# B&R Automation Studio project X20CP1382
Automation Studio 4.12.2.93; technology packages: mappView 5.16.1

## Configuration Config1

CPU X20CP1382, AutomationRuntime D4.83, Build 4.1.2, Safety 0.0, Vc V4.72.3

### Task classes (Cpu.sw)
```
Cyclic#4:
  Program1 <- Program1.prg
  Program <- Program.prg
  Zufall <- Zufall.prg
Binaries: FWRules, mvLoader, udbdef, TCData, iomap, sysconf, asfw, User, arconfig, ashwd, Role, ashwac
Libraries: standard, asieccon, astime, arssl, runtime, fileio
```

### Hardware
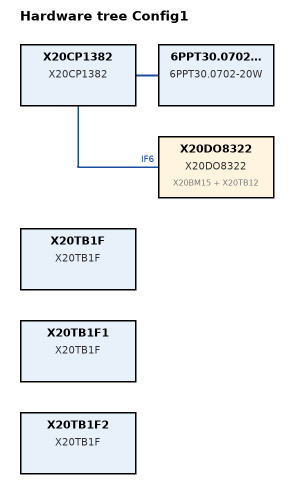
```
6PPT30.0702-20W : 6PPT30.0702-20W v1.3.5.0  [ETH1 -> X20CP1382.IF2 [Cable Type=PowerlinkCable, Length=10, Version=1.0.0.3]]
  Terminal = true
  Mode = Manual
  InternetAddress = 192.168.10.4
  Subnetmask = 255.255.255.0
  PasswordVNC = 
  PasswordCIFS = 
  PasswordService = 
  VncKeyMappingFile = VC\6PPT30.0702-20W.dis
X20BM15 : X20BM15 v1.1.0.0  [X2X1 -> X20CP1382.IF6 (NodeNumber=1)]
X20CP1382 : X20CP1382 v1.14.0.0  [X1 -> X1.SL; X2 -> X2.SL; X3 -> X3.SL]
  Module X1 (Type=X1, Virtual=true, Version=1.14.0.0)
    Connection (Connector=SS1, TargetModule=X20TB1F, TargetConnector=SS)
    Connection (Connector=SL, TargetModule=X20CP1382, TargetConnector=X1)
  Module X2 (Type=X2, Virtual=true, Version=1.14.0.0)
    Connection (Connector=SS1, TargetModule=X20TB1F1, TargetConnector=SS)
    Connection (Connector=SL, TargetModule=X20CP1382, TargetConnector=X2)
  Module X3 (Type=X3, Virtual=true, Version=1.14.0.0)
    Connection (Connector=SS1, TargetModule=X20TB1F2, TargetConnector=SS)
    Connection (Connector=SL, TargetModule=X20CP1382, TargetConnector=X3)
  Connector IF2:
    ActivateDevice = 1
    Mode = Manual
    InternetAddress = 192.168.10.5
    SubnetMask = 255.255.255.0
    ActivateSnmp = 2
  ConfigurationID = X20CP1382_Config1
  Simulation = 1
  ActivateOpcUa = 1
  OpcUaInformationModels_PV_Version = 1
X20DO8322 : X20DO8322 v1.5.0.0  [SS1 -> X20TB12a.SS; SL -> X20BM15.SL1]
X20TB12a : X20TB12 v1.0.0.0
X20TB1F : X20TB1F v1.0.0.0
X20TB1F1 : X20TB1F v1.0.0.0
X20TB1F2 : X20TB1F v1.0.0.0
```

### IoMap.iom - X20CP1382/IoMap.iom
```iecst
VAR_CONFIG
	::Program:directionThreadmillleft_DO AT %QX."X3".DigitalOutput12;
	::pumpeBig1_DO AT %QX."X3".DigitalOutput01;
	::pumpeBig2_DO AT %QX."X3".DigitalOutput02;
	::pumpeBig3_DO AT %QX."X3".DigitalOutput03;
	::pumpeBig4_DO AT %QX."X3".DigitalOutput04;
	::pumpeSmall1_DO AT %QX."X3".DigitalOutput05;
	::pumpeSmall2_DO AT %QX."X3".DigitalOutput06;
	::pumpeSmall3_DO AT %QX."X3".DigitalOutput07;
	::pumpeSmall4_DO AT %QX."X3".DigitalOutput08;
	::pumpeSmall5_DO AT %QX."X3".DigitalOutput09;
	::Program:directionTreadmillright_DO AT %QX."X3".DigitalOutput11;
	::pumpeSmall6_DO AT %QX."X3".DigitalOutput10;
	::Program:inductiveSensorBecherspender_DI AT %IX."X2".DigitalInput01;
	::Program:inductiveSensorEisstation_DI AT %IX."X2".DigitalInput02;
	::Program:inductiveSensorZitronenspende_DI AT %IX."X2".DigitalInput03;
	::Program:inductiveSensorCocktailmixer_DI AT %IX."X2".DigitalInput04;
	::Program:inductiveSensorBecherausgabe_DI AT %IX."X2".DigitalInput05;
	::Program:bechererkennungSpender_DI AT %IX."X2".DigitalInput06;
	::Program:bechererkennungAusgabe_DI AT %IX."X2".DigitalInput07;
	::Program:BecherspenderAktivieren_DO AT %QX."X20DO8322".DigitalOutput01;
	::Program:eisspenderAktivieren_DO AT %QX."X20DO8322".DigitalOutput02;
	::ERROR_DI AT %IX."X2".DigitalInput08 INVERSE;
	::Program:zitronenspenderAktivieren_DO AT %QX."X20DO8322".DigitalOutput03;
	::Program:lichtschrankeEismaschine_DI AT %IX."X2".DigitalInput10;
	::Program:endlagenschArmCocktailStation_DI AT %IX."X2".DigitalInput09;
	::Program:armCocktailstation_DO AT %QX."X20DO8322".DigitalOutput04;
END_VAR
```

## Logical view

### Global.var - Globale Variablen
```iecst
VAR
	pumpeBig1_DO : BOOL;
	pumpeBig2_DO : BOOL;
	pumpeBig3_DO : BOOL;
	pumpeBig4_DO : BOOL;
	pumpeSmall1_DO : BOOL;
	pumpeSmall2_DO : BOOL;
	pumpeSmall3_DO : BOOL;
	pumpeSmall4_DO : BOOL;
	pumpeSmall5_DO : BOOL;
	pumpeSmall6_DO : BOOL;
	cocktailFinished_var : BOOL;
	cocktailChosen_var : BOOL := FALSE; (*Gibt an, ob ein Cocktail gewählt wurde*)
	counterCocktailmixer_var : UDINT := 0; (*Wenn Station erstes mal angefahren wird Cocktail ausgegeben*)
	reingigunsmodus_var : BOOL := FALSE; (*Gibt an, ob die Reinigung aktiviert wurde*)
	cocktail_started : BOOL; (*Triggert die Pumpen für den aktuellen Cocktail*)
	ERROR_DI : BOOL := FALSE; (*STOPPT SPS KOMPLETT*)
	zufallscocktailAktivieren : BOOL;
	zutat_JaNein_ok : ARRAY[1..10] OF BOOL; (*Array mit Info, ob Zutat verwendet wird oder nicht*)
	zutat_Menge_ok : ARRAY[1..10] OF UINT; (*Array mit Info, wie viele ml der Zutat rein sollen*)
	zufallscocktail_var : BOOL := FALSE;
END_VAR
```

### Program Logical/Program (IEC)

#### Variables.var
```iecst
VAR
	armCocktailstation_DO : BOOL := FALSE; (*Gibt Signal für Arm nach oben und unten*)
	stationPercentage_var : USINT := 0; (*gibt in der Visualisierung den aktuellen Progress in % aus*)
	resetToStart_var : BOOL := TRUE; (*Fährt wieder an den Start*)
	passwordVisu_st : WSTRING[40] := "student"; (*Passwort 'student42'*)
	passwordVisuCorrect_var : BOOL := FALSE; (*gibt 1 aus wenn passwort stimmt*)
	lichtschrankeEismaschine_DI : BOOL := FALSE; (*Reagiert auf den Arduino mit der Lichtschranke*)
	inductiveSensorZitronenspende_DI : BOOL := FALSE; (*Station Zitronenspender Sensorerkennung*)
	inductiveSensorEisstation_DI : BOOL := FALSE; (*Station Eisstation Sensorerkennung*)
	inductiveSensorCocktailmixer_DI : BOOL := FALSE; (*Station Cocktailmixer Sensorenerkennung*)
	inductiveSensorBecherspender_DI : BOOL := FALSE; (*Station Becherspender Sensorerkennung*)
	inductiveSensorBecherausgabe_DI : BOOL := FALSE; (*Station Becherausgabe Sensorenerkennung*)
	hilfsDelayArmCocktailStation_var : UDINT := 0; (*hilft mit dem Timing für den Arm, damit die Pumpen sicher abgeschalten haben für bewegung*)
	resetCounter_var : USINT := 0; (*lässt wagen erstmal nach rechts und danach nach links fahren*)
	endlagenschArmCocktailStation_DI : BOOL := FALSE; (*Zeigt an, ob becher unter dem Endlagenschalter ist*)
	eisspenderAktivieren_DO : BOOL := FALSE; (*Aktiviert den Eisspender --> Arduino*)
	goToMainpage_var : BOOL := FALSE; (*Geht wieder zurück auf die Hauptseite*)
	directionThreadmill_right_var : BOOL := FALSE; (*Kann nur im Reinigunsprogramm gesetzt werden*)
	bechererkennungAusgabe_DI : BOOL := TRUE; (*Wenn endlageschalter nicht gedrückt ist, Becher entnommen*)
	bechererkennungSpender_DI : BOOL := FALSE; (*Wenn endlageschalter gedrückt, Becher in Halterung*)
	BecherspenderAktivieren_DO : BOOL := FALSE; (*Aktiviert Becherspender --> Arduino *)
	directionTreadmillright_DO : BOOL := FALSE; (*Steuert das Laufband nach rechts*)
	counterBecherspender_var : USINT := 0; (*Setzt die Zeit für die Sation Becherspender*)
	counterEisstation_var : UINT := 0; (*Setzt die Zeit für die Sation Eisstation*)
	counterBecherentnahme_var : USINT := 0; (*Setzt die Zeit für die Station Becherentnahme*)
	currentBecherausgabeState_var : USINT := 0; (*Switch Case Becherausgabe*)
	currentCocktialState_var : USINT := 0; (*Läuft die einzelnen unterstationen im Cocktailmixer ab*)
	currentStation_var : USINT := 0; (*Läuft die einzelnen Sationen ab*)
	delayCocktailStation_var : USINT := 0; (*Ein Delay nach dem Cocktaileinfüllen*)
	directionThreadmillleft_DO : BOOL := FALSE; (*Steuert das Laufband nach links*)
	directionThreadmill_left_var : BOOL := FALSE; (*Kann nur im Reinigunsprogramm gesetzt werden*)
	counterZitronenspender_var : USINT := 0; (*Setzt die Zeit für die Sation Zitronenspender*)
	zitronenspenderAktivieren_DO : BOOL := FALSE; (*Aktiviert Zitronenspender --> Arduino *)
END_VAR
VAR CONSTANT
	stationBecherentnahme_var : USINT := 4; (*Station Becherentnahme als Festwerte*)
	stationBecherspender_var : USINT := 0; (*Station Becherspender als Festwerte*)
	stationCocktailmixer_var : USINT := 3; (*Station Cocktailmixer als Festwerte*)
	stationEismaschine_var : USINT := 1; (*Station Eismaschine als Festwerte*)
END_VAR
VAR
	hilfsCounterEismaschine_var : UDINT := 0; (*Zählt einen Delay ein, damit der Wagen nicht direkt weiterfährt, wenn die Eiswürfel kommen*)
	deactivatesAllPumps_var : BOOL := FALSE; (*Kann im Reinigunsprogramm aktiviert werden und schaltet alle Pumpen AUS*)
	activatesAllPumps_var : BOOL := FALSE; (*Kann im Reinigungsprogramm aktiviert werden und schaltet alle Pumpen AN*)
END_VAR
VAR CONSTANT
	stationZitronenspender_var : USINT := 2; (*Station Zitronenspender als Festwert*)
END_VAR
```

#### Cyclic.st
```iecst
PROGRAM _CYCLIC
	// Visualisierungs Passworteingabe
	IF passwordVisu_st = "student42" THEN
		passwordVisuCorrect_var := TRUE;
	ELSE
		passwordVisuCorrect_var := FALSE;
	END_IF

	IF ERROR_DI = TRUE THEN
		// ON ERROR STOPPT ALLE PUMPEN DIREKT
		pumpeBig1_DO := FALSE;
		pumpeBig2_DO := FALSE;
		pumpeBig3_DO := FALSE;
		pumpeBig4_DO := FALSE;
		pumpeSmall1_DO := FALSE;
		pumpeSmall2_DO := FALSE;
		pumpeSmall3_DO := FALSE;
		pumpeSmall4_DO := FALSE;
		pumpeSmall5_DO := FALSE;
		pumpeSmall6_DO := FALSE;

		directionTreadmillright_DO := FALSE;
		directionThreadmillleft_DO := FALSE;
	ELSE
		// Reinigungsprogramm
		IF reingigunsmodus_var = TRUE THEN
			IF directionThreadmill_left_var = TRUE THEN
				directionThreadmillleft_DO := 0;
				directionTreadmillright_DO := 1;
			END_IF
			IF directionThreadmill_right_var = TRUE THEN
				directionThreadmillleft_DO := 1;
				directionTreadmillright_DO := 0;
			END_IF
			IF directionThreadmill_right_var = FALSE AND directionThreadmill_left_var = FALSE THEN
				directionThreadmillleft_DO := 0;
				directionTreadmillright_DO := 0;
			END_IF

			IF activatesAllPumps_var = TRUE THEN
				activatesAllPumps_var := FALSE;
				pumpeBig1_DO := TRUE;
				pumpeBig2_DO := TRUE;
				pumpeBig3_DO := TRUE;
				pumpeBig4_DO := TRUE;
				pumpeSmall1_DO := TRUE;
				pumpeSmall2_DO := TRUE;
				pumpeSmall3_DO := TRUE;
				pumpeSmall4_DO := TRUE;
				pumpeSmall5_DO := TRUE;
				pumpeSmall6_DO := TRUE;
			END_IF

			IF deactivatesAllPumps_var = TRUE THEN
				deactivatesAllPumps_var := FALSE;
				pumpeBig1_DO := FALSE;
				pumpeBig2_DO := FALSE;
				pumpeBig3_DO := FALSE;
				pumpeBig4_DO := FALSE;
				pumpeSmall1_DO := FALSE;
				pumpeSmall2_DO := FALSE;
				pumpeSmall3_DO := FALSE;
				pumpeSmall4_DO := FALSE;
				pumpeSmall5_DO := FALSE;
				pumpeSmall6_DO := FALSE;
			END_IF

		ELSE
			CASE currentStation_var OF
				stationBecherspender_var:
					// Setzt Website wieder auf Hauptseite nach erfolgten Durchlauf
					IF inductiveSensorBecherspender_DI = FALSE OR counterBecherspender_var > 0 THEN
						IF currentBecherausgabeState_var = 3 THEN
							goToMainpage_var := TRUE;
							resetCounter_var := 0;
							currentBecherausgabeState_var := 0;
						END_IF

						directionThreadmillleft_DO := 0;
						counterBecherentnahme_var := 0;
						IF cocktailChosen_var = TRUE THEN
							goToMainpage_var := FALSE;
							currentBecherausgabeState_var := 0;
							counterBecherspender_var := counterBecherspender_var + 1;

							stationPercentage_var := 10;

							IF counterBecherspender_var = 1 THEN
								BecherspenderAktivieren_DO := TRUE;
							ELSE
								BecherspenderAktivieren_DO := FALSE;
							END_IF

							IF bechererkennungSpender_DI = TRUE THEN
								directionTreadmillright_DO := 1;
								currentStation_var := currentStation_var + 1;
								BecherspenderAktivieren_DO := FALSE;
								stationPercentage_var := 20;
							END_IF
						END_IF
					END_IF

				stationEismaschine_var:
					IF inductiveSensorEisstation_DI = FALSE OR counterEisstation_var > 0 THEN
						directionTreadmillright_DO := 0;
						counterBecherspender_var := 0;
						counterEisstation_var := counterEisstation_var + 1;
						stationPercentage_var := 30;

						// 300 ms impuls for Arduino bei Anfahren der Station
						IF counterEisstation_var < 4 THEN
							eisspenderAktivieren_DO := TRUE;
						ELSE
							eisspenderAktivieren_DO := FALSE;
						END_IF

						// Wenn die Lichtschrankenrückmeldung kommt
						IF lichtschrankeEismaschine_DI = TRUE AND hilfsCounterEismaschine_var = 0 AND counterEisstation_var > 5 THEN
							hilfsCounterEismaschine_var := counterEisstation_var + 30;
						END_IF

						// Wenn der Wagen an der Station für 15 Sekunden steht oder das Signal vom Arduino kommt, das Lichtschranke ausgelöst wurde
						IF counterEisstation_var > 3000 OR hilfsCounterEismaschine_var <= counterEisstation_var AND hilfsCounterEismaschine_var <> 0 THEN
							directionTreadmillright_DO := 1;
							currentStation_var := currentStation_var + 1;
							stationPercentage_var := 40;
						END_IF
					END_IF

				stationZitronenspender_var:
					IF inductiveSensorZitronenspende_DI = FALSE OR counterZitronenspender_var > 0 THEN
						hilfsCounterEismaschine_var := 0;
						directionTreadmillright_DO := 0;
						counterEisstation_var := 0;
						counterZitronenspender_var := counterZitronenspender_var + 1;
						stationPercentage_var := 50;

						// 400 ms impuls for arduino
						IF counterZitronenspender_var < 4 THEN
							zitronenspenderAktivieren_DO := TRUE;
						ELSE
							zitronenspenderAktivieren_DO := FALSE;
						END_IF

						IF counterZitronenspender_var > 50 THEN
							directionTreadmillright_DO := 1;
							currentStation_var := currentStation_var + 1;
							stationPercentage_var := 60;
						END_IF
					END_IF

				stationCocktailmixer_var:
					IF inductiveSensorCocktailmixer_DI = FALSE OR counterCocktailmixer_var > 0 THEN
						directionTreadmillright_DO := 0;
						counterZitronenspender_var := 0;
						counterCocktailmixer_var := counterCocktailmixer_var + 1;

						CASE currentCocktialState_var OF
							0:
								// Arm fährt runter --> Signal Arduino
								IF counterCocktailmixer_var > 3 THEN
									armCocktailstation_DO := TRUE;
									currentCocktialState_var := currentCocktialState_var + 1;
									stationPercentage_var := 70;
								END_IF
							1:
								// Setzt Arduino Signal wieder auf 0
								IF counterCocktailmixer_var > 7 THEN;
									armCocktailstation_DO := FALSE;
									currentCocktialState_var := currentCocktialState_var + 1;
								END_IF

							2:
								// Startet Cocktail, wenn Endlagenschalter Anschlägt
								IF counterCocktailmixer_var >= 30 AND endlagenschArmCocktailStation_DI = TRUE THEN
									cocktail_started := FALSE;
									currentCocktialState_var := currentCocktialState_var + 1;
								END_IF
							3:
								//	IF cocktailFinished_var = TRUE THEN
								IF counterCocktailmixer_var >= 50 AND pumpeBig1_DO = 0 AND pumpeBig2_DO = 0 AND pumpeBig3_DO = 0 AND pumpeBig4_DO = 0 AND pumpeSmall1_DO = 0 AND pumpeSmall2_DO = 0 AND pumpeSmall3_DO = 0 AND pumpeSmall4_DO = 0 AND  pumpeSmall5_DO = 0 AND  pumpeSmall6_DO = 0 THEN
									stationPercentage_var := 80;
									cocktailFinished_var := TRUE;

									hilfsDelayArmCocktailStation_var := counterCocktailmixer_var + 5;
									currentCocktialState_var := currentCocktialState_var + 1;
								END_IF
							4:
								// Delay nach dem die Pumpen abgeschalten haben 500ms
								IF counterCocktailmixer_var >= hilfsDelayArmCocktailStation_var AND armCocktailstation_DO = FALSE THEN
									armCocktailstation_DO := TRUE;
									hilfsDelayArmCocktailStation_var :=  counterCocktailmixer_var + 4;
									currentCocktialState_var := currentCocktialState_var + 1;
								END_IF
							5:
								// 400 ms Signal auf den Ausgang beenden
								IF counterCocktailmixer_var >= hilfsDelayArmCocktailStation_var AND armCocktailstation_DO = TRUE THEN
									stationPercentage_var := 90;
									armCocktailstation_DO := FALSE;
									hilfsDelayArmCocktailStation_var := counterCocktailmixer_var + 16;
									currentCocktialState_var := currentCocktialState_var + 1;
								END_IF
							6:
								// geht zur nächsten Station nachdem der arm 1.6 Sekunden Zeit hatte hochzufahren
								IF 	counterCocktailmixer_var >= hilfsDelayArmCocktailStation_var AND stationPercentage_var = 90 THEN
									directionTreadmillright_DO := TRUE;
									currentStation_var := currentStation_var + 1;
									currentCocktialState_var := 0;
								END_IF
						END_CASE
					END_IF

				stationBecherentnahme_var:
					CASE currentBecherausgabeState_var OF
						0: // Stoppt an Station
							IF inductiveSensorBecherausgabe_DI = FALSE OR bechererkennungAusgabe_DI = TRUE THEN
								counterCocktailmixer_var := 0;
								currentBecherausgabeState_var := 1;
								cocktailFinished_var := 0;
								stationPercentage_var := 100;
								directionTreadmillright_DO := 0;
								delayCocktailStation_var := 0;
							END_IF

						1:// Wenn Becher steht
							// drei Sekunden verzögerung zum verlässlichen erkennen des Endlagenschalters
							IF counterBecherentnahme_var >= 30 THEN
								// Erkennt wenn Becher Ausgegeben wurde --> Wird als zweites ausgeführt
								IF bechererkennungAusgabe_DI = FALSE THEN
									currentBecherausgabeState_var := 2;
								END_IF
							ELSE
								counterBecherentnahme_var := counterBecherentnahme_var + 1;
							END_IF

						2:
							// Zählt Für Verzögerung beim herausnehmen
							IF counterBecherentnahme_var > 0 THEN
								counterBecherentnahme_var := counterBecherentnahme_var + 1;
							END_IF

							// Fährt mit verzögerung wieder zum Start
							IF counterBecherentnahme_var >= 60 THEN
								directionTreadmillright_DO := 0;
								directionThreadmillleft_DO := 1;
								currentStation_var := 0;
								cocktailChosen_var := FALSE;
								currentBecherausgabeState_var := 3;
							END_IF
					END_CASE
			END_CASE
		END_IF

		// Zurücksetzen auf Start
		IF resetToStart_var = TRUE THEN
			IF resetCounter_var < 10 THEN
				resetCounter_var := resetCounter_var + 1;
				pumpeBig1_DO := FALSE;
				pumpeBig2_DO := FALSE;
				pumpeBig3_DO := FALSE;
				pumpeBig4_DO := FALSE;
				pumpeSmall1_DO := FALSE;
				pumpeSmall2_DO := FALSE;
				pumpeSmall3_DO := FALSE;
				pumpeSmall4_DO := FALSE;
				pumpeSmall5_DO := FALSE;
				pumpeSmall6_DO := FALSE;

				counterBecherspender_var := 0;
				counterEisstation_var := 0;
				counterZitronenspender_var := 0;
				counterCocktailmixer_var := 0;

				directionThreadmillleft_DO := 0;

				// Fährt nich weiter, wenn hinten der Taster gedrückt wird
				IF bechererkennungAusgabe_DI = FALSE THEN
					directionTreadmillright_DO := 1;
				ELSE
					directionTreadmillright_DO := 0;
				END_IF
			ELSE
				directionTreadmillright_DO := 0;
				currentStation_var := 4;
				currentBecherausgabeState_var := 2;
				counterBecherentnahme_var := 100;

				resetToStart_var := FALSE;
			END_IF
		END_IF
	END_IF
END_PROGRAM
```

#### Init.st
```iecst
PROGRAM _INIT

END_PROGRAM
```

### Program Logical/Program1 (IEC)

#### Types.typ
```iecst
TYPE
	cocktail_name :
		(
		wodka_cola,
		kirschcola,
		testcocktail,
		wodka_osaft,
		gruenewiese,
		angelblue,
		brassmonkey,
		kiba,
		rumcola,
		gintonic,
		bluelagoon,
		cola,
		osaft,
		banane,
		tonic,
		sprite,
		zufallscocktail
		);
END_TYPE
```

#### Variables.var
```iecst
VAR
	cocktail_var : cocktail_name;
	cocktail_start : BOOL;
	TOF_01 : TOF;
	TOF_02 : TOF;
	TOF_03 : TOF;
	TOF_04 : TOF;
	TOF_05 : TOF;
	TOF_06 : TOF;
	TOF_07 : TOF;
	TOF_08 : TOF;
	TOF_09 : TOF;
	TOF_10 : TOF;
	pumptime_01 : TIME;
	pumptime_02 : TIME;
	pumptime_03 : TIME;
	pumptime_04 : TIME;
	pumptime_05 : TIME;
	pumptime_06 : TIME;
	pumptime_07 : TIME;
	pumptime_08 : TIME;
	pumptime_09 : TIME;
	pumptime_10 : TIME;
	ml_wodkacola_wodka : UINT := 50;
	ml_wodkacola_cola : UINT := 250;
	ml_wodkaosaft_osaft : UINT := 250;
	ml_wodkaosaft_wodka : UINT := 50;
	ml_rumcola_cola : UINT := 250;
	ml_rumcola_rum : UINT := 50;
	ml_kirschcola_cola : UINT := 210;
	ml_kirschcola_kirsch : UINT := 90;
	ml_gruenewiese_osaft : UINT := 220;
	ml_gruenewiese_bc : UINT := 80;
	ml_angelblue_sprite : UINT := 200;
	ml_angelblue_bc : UINT := 70;
	ml_angelblue_wodka : UINT := 30;
	ml_brassmonkey_osaft : UINT := 240;
	ml_brassmonkey_wodka : UINT := 30;
	ml_brassmonkey_rum : UINT := 30;
	ml_kiba_banane : UINT := 210;
	ml_kiba_kirsch : UINT := 90;
	ml_gintonic_tonic : UINT := 250;
	ml_gintonic_gin : UINT := 50;
	ml_osaft : UINT := 300;
	ml_cola : UINT := 300;
	ml_banane : UINT := 300;
	ml_tonic : UINT := 300;
	ml_sprite : UINT := 300;
	ml_bluelagoon_sprite : UINT := 220;
	ml_bluelagoon_bc : UINT := 80;
	wodka_cola_var : BOOL := FALSE;
	kirschcola_var : BOOL := FALSE;
	testcocktail_var : BOOL := FALSE;
	gruenewiese_var : BOOL := FALSE;
	brassmonkey_var : BOOL := FALSE;
	angelblue_var : BOOL := FALSE;
	kiba_var : BOOL := FALSE;
	rumcola_var : BOOL := FALSE;
	gintonic_var : BOOL := FALSE;
	wodka_osaft_var : BOOL := FALSE;
	osaft_var : BOOL := FALSE;
	cola_var : BOOL := FALSE;
	banane_var : BOOL := FALSE;
	tonic_var : BOOL := FALSE;
	sprite_var : BOOL := FALSE;
	bluelagoon_var : BOOL := FALSE;
END_VAR
VAR RETAIN
	Anzahl_Cocktails : ARRAY[0..19] OF INT := [20(0)];
END_VAR
```

#### Cyclic.st
```iecst
PROGRAM _CYCLIC

	IF (cocktail_start = FALSE AND cocktail_started = FALSE) THEN
		cocktail_start := TRUE;
	END_IF

	// Wenn Reinigungsprogramm aktiviert ist, soll kein Cocktail gemacht werden
	IF reingigunsmodus_var = FALSE AND ERROR_DI = FALSE THEN
		CASE cocktail_var OF
			wodka_cola:
				pumptime_01 :=	UINT_TO_TIME(ml_wodkacola_cola)*108;
				pumptime_02 :=	UINT_TO_TIME(ml_wodkacola_wodka)*330;

				TOF_01(IN:= cocktail_start , PT:= pumptime_01 );
				pumpeBig2_DO:=TOF_01.Q;

				TOF_02(IN:= cocktail_start , PT:= pumptime_02 );
				pumpeSmall3_DO:=TOF_02.Q;

			rumcola:
				pumptime_01 :=	UINT_TO_TIME(ml_rumcola_cola)*108;
				pumptime_02 :=	UINT_TO_TIME(ml_rumcola_rum)*420;

				TOF_01(IN:= cocktail_start , PT:= pumptime_01 );
				pumpeBig2_DO:=TOF_01.Q;

				TOF_02(IN:= cocktail_start , PT:= pumptime_02 );
				pumpeSmall2_DO:=TOF_02.Q;

			kirschcola:
				pumptime_01 :=	UINT_TO_TIME(ml_kirschcola_cola)*108;
				pumptime_02 :=	UINT_TO_TIME(ml_kirschcola_kirsch)*390;

				TOF_01(IN:= cocktail_start , PT:= pumptime_01 );
				pumpeBig2_DO:=TOF_01.Q;

				TOF_02(IN:= cocktail_start , PT:= pumptime_02 );
				pumpeSmall5_DO:=TOF_02.Q;

			gruenewiese:
				pumptime_01 :=	UINT_TO_TIME(ml_gruenewiese_osaft)*118;
				pumptime_02 :=	UINT_TO_TIME(ml_gruenewiese_bc)*350;

				TOF_01(IN:= cocktail_start , PT:= pumptime_01 );
				pumpeBig4_DO:=TOF_01.Q;

				TOF_02(IN:= cocktail_start , PT:= pumptime_02 );
				pumpeSmall6_DO:=TOF_02.Q;

			angelblue:
				pumptime_01 :=	UINT_TO_TIME(ml_angelblue_sprite)*111;
				pumptime_02 :=	UINT_TO_TIME(ml_angelblue_bc)*350;
				pumptime_03 := UINT_TO_TIME(ml_angelblue_wodka)*330;

				TOF_01(IN:= cocktail_start , PT:= pumptime_01 );
				pumpeBig1_DO:=TOF_01.Q;

				TOF_02(IN:= cocktail_start , PT:= pumptime_02 );
				pumpeSmall6_DO:=TOF_02.Q;

				TOF_03(IN:= cocktail_start , PT:= pumptime_03 );
				pumpeSmall3_DO:=TOF_03.Q;

			brassmonkey:
				pumptime_01 :=	UINT_TO_TIME(ml_brassmonkey_osaft)*118;
				pumptime_02 :=	UINT_TO_TIME(ml_brassmonkey_rum)*420;
				pumptime_03 := UINT_TO_TIME(ml_angelblue_wodka)*330;

				TOF_01(IN:= cocktail_start , PT:= pumptime_01 );
				pumpeBig4_DO:=TOF_01.Q;

				TOF_02(IN:= cocktail_start , PT:= pumptime_02 );
				pumpeSmall2_DO:=TOF_02.Q;

				TOF_03(IN:= cocktail_start , PT:= pumptime_03 );
				pumpeSmall3_DO:=TOF_03.Q;

			wodka_osaft:
				pumptime_01 :=	UINT_TO_TIME(ml_wodkaosaft_osaft)*118;
				pumptime_02 :=	UINT_TO_TIME(ml_wodkaosaft_wodka)*330;

				TOF_01(IN:= cocktail_start , PT:= pumptime_01 );
				pumpeBig4_DO:=TOF_01.Q;

				TOF_02(IN:= cocktail_start , PT:= pumptime_02 );
				pumpeSmall3_DO:=TOF_02.Q;

			testcocktail:
				pumptime_01 :=	T#2s;
				pumptime_02 :=	T#2s;

				TOF_01(IN:= cocktail_start , PT:= pumptime_01 );
				pumpeBig4_DO:=TOF_01.Q;

				TOF_02(IN:= cocktail_start , PT:= pumptime_02 );
				pumpeSmall3_DO:=TOF_02.Q;

			kiba:
				pumptime_01 :=	UINT_TO_TIME(ml_kiba_banane)*105;
				pumptime_02 :=	UINT_TO_TIME(ml_kiba_kirsch)*390;

				TOF_01(IN:= cocktail_start , PT:= pumptime_01 );
				pumpeBig3_DO:=TOF_01.Q;

				TOF_02(IN:= cocktail_start , PT:= pumptime_02 );
				pumpeSmall5_DO:=TOF_02.Q;

			gintonic:
				pumptime_01 :=	UINT_TO_TIME(ml_gintonic_tonic)*390;
				pumptime_02 :=	UINT_TO_TIME(ml_gintonic_gin)*300;

				TOF_01(IN:= cocktail_start , PT:= pumptime_01 );
				pumpeSmall1_DO:=TOF_01.Q;

				TOF_02(IN:= cocktail_start , PT:= pumptime_02 );
				pumpeSmall4_DO:=TOF_02.Q;

			bluelagoon:
				pumptime_01 :=	UINT_TO_TIME(ml_bluelagoon_sprite)*111;
				pumptime_02 :=	UINT_TO_TIME(ml_bluelagoon_bc)*350;

				TOF_01(IN:= cocktail_start , PT:= pumptime_01 );
				pumpeBig1_DO:=TOF_01.Q;

				TOF_02(IN:= cocktail_start , PT:= pumptime_02 );
				pumpeSmall6_DO:=TOF_02.Q;

			zufallscocktail:
				pumptime_01 :=	UINT_TO_TIME(zutat_Menge_ok[1])*111;
				pumptime_02 :=	UINT_TO_TIME(zutat_Menge_ok[2])*108;
				pumptime_03 :=	UINT_TO_TIME(zutat_Menge_ok[3])*105;
				pumptime_02 :=	UINT_TO_TIME(zutat_Menge_ok[4])*118;
				pumptime_05 :=	UINT_TO_TIME(zutat_Menge_ok[5])*390;
				pumptime_06 :=	UINT_TO_TIME(zutat_Menge_ok[6])*420;
				pumptime_07 :=	UINT_TO_TIME(zutat_Menge_ok[7])*330;
				pumptime_08 :=	UINT_TO_TIME(zutat_Menge_ok[8])*300;
				pumptime_09 :=	UINT_TO_TIME(zutat_Menge_ok[9])*390;
				pumptime_10 :=	UINT_TO_TIME(zutat_Menge_ok[10])*350;

				IF zutat_JaNein_ok[1] = TRUE THEN
					TOF_01(IN:= cocktail_start , PT:= pumptime_01 );
					pumpeBig1_DO:=TOF_01.Q;
				END_IF
				IF zutat_JaNein_ok[2] = TRUE THEN
					TOF_02(IN:= cocktail_start , PT:= pumptime_02 );
					pumpeBig2_DO:=TOF_02.Q;
				END_IF
				IF zutat_JaNein_ok[3] = TRUE THEN
					TOF_03(IN:= cocktail_start , PT:= pumptime_03 );
					pumpeBig3_DO:=TOF_03.Q;
				END_IF
				IF zutat_JaNein_ok[4] = TRUE THEN
					TOF_04(IN:= cocktail_start , PT:= pumptime_04 );
					pumpeBig4_DO:=TOF_04.Q;
				END_IF
				IF zutat_JaNein_ok[5] = TRUE THEN
					TOF_05(IN:= cocktail_start , PT:= pumptime_05 );
					pumpeSmall1_DO:=TOF_05.Q;
				END_IF
				IF zutat_JaNein_ok[6] = TRUE THEN
					TOF_06(IN:= cocktail_start , PT:= pumptime_06 );
					pumpeSmall2_DO:=TOF_06.Q;
				END_IF
				IF zutat_JaNein_ok[7] = TRUE THEN
					TOF_07(IN:= cocktail_start , PT:= pumptime_07 );
					pumpeSmall3_DO:=TOF_07.Q;
				END_IF
				IF zutat_JaNein_ok[8] = TRUE THEN
					TOF_08(IN:= cocktail_start , PT:= pumptime_08 );
					pumpeSmall4_DO:=TOF_08.Q;
				END_IF
				IF zutat_JaNein_ok[9] = TRUE THEN
					TOF_09(IN:= cocktail_start , PT:= pumptime_09 );
					pumpeSmall5_DO:=TOF_09.Q;
				END_IF
				IF zutat_JaNein_ok[10] = TRUE THEN
					TOF_10(IN:= cocktail_start , PT:= pumptime_10 );
					pumpeSmall6_DO:=TOF_10.Q;
				END_IF

			osaft:
				pumptime_01 :=	UINT_TO_TIME(ml_osaft)*118;

				TOF_01(IN:= cocktail_start , PT:= pumptime_01 );
				pumpeBig4_DO:=TOF_01.Q;
			cola:
				pumptime_01 :=	UINT_TO_TIME(ml_cola)*108;

				TOF_01(IN:= cocktail_start , PT:= pumptime_01 );
				pumpeBig2_DO:=TOF_01.Q;
			banane:
				pumptime_01 :=	UINT_TO_TIME(ml_banane)*105;

				TOF_01(IN:= cocktail_start , PT:= pumptime_01 );
				pumpeBig3_DO:=TOF_01.Q;
			tonic:
				pumptime_01 :=	UINT_TO_TIME(ml_tonic)*390;

				TOF_01(IN:= cocktail_start , PT:= pumptime_01 );
				pumpeSmall1_DO:=TOF_01.Q;
			sprite:
				pumptime_01 :=	UINT_TO_TIME(ml_sprite)*111;

				TOF_01(IN:= cocktail_start , PT:= pumptime_01 );
				pumpeBig1_DO:=TOF_01.Q;

		END_CASE
	END_IF
	// IF Cocktail was chosen in the visualisation --> Cocktailchosen == True
	IF wodka_cola_var = 1 OR kirschcola_var = 1 OR testcocktail_var = 1 OR wodka_osaft_var = 1 OR gruenewiese_var = 1 OR angelblue_var = 1 OR brassmonkey_var = 1 OR kiba_var = 1 OR rumcola_var = 1 OR gintonic_var = 1 OR bluelagoon_var = 1 OR osaft_var = 1 OR cola_var = 1 OR banane_var = 1 OR tonic_var = 1 OR sprite_var = 1 OR zufallscocktail_var = 1 THEN
		cocktailChosen_var := TRUE;
	END_IF

	IF (cocktail_start = TRUE AND cocktail_started = FALSE) THEN
		cocktail_start := FALSE;
		cocktail_started := TRUE;

		// Variable, dass Cocktail beendet wurde
		cocktailFinished_var := TRUE;
	END_IF

	// Setzt den Schalter zurück
	IF wodka_cola_var = TRUE THEN
		cocktail_var := wodka_cola;
		wodka_cola_var := FALSE;
		Anzahl_Cocktails [wodka_cola] := Anzahl_Cocktails [wodka_cola] + 1;
	END_IF
	IF kirschcola_var = TRUE THEN
		cocktail_var := kirschcola;
		kirschcola_var := FALSE;
		Anzahl_Cocktails [kirschcola] := Anzahl_Cocktails [kirschcola] + 1;
	END_IF
	IF testcocktail_var = TRUE THEN
		cocktail_var := testcocktail;
		testcocktail_var := FALSE;
		Anzahl_Cocktails [testcocktail] := Anzahl_Cocktails [testcocktail] + 1;
	END_IF
	IF wodka_osaft_var = TRUE THEN
		cocktail_var := wodka_osaft;
		wodka_osaft_var := FALSE;
		Anzahl_Cocktails [wodka_osaft] := Anzahl_Cocktails [wodka_osaft] + 1;
	END_IF
	IF gruenewiese_var = TRUE THEN
		cocktail_var := gruenewiese;
		gruenewiese_var := FALSE;
		Anzahl_Cocktails [gruenewiese] := Anzahl_Cocktails [gruenewiese] + 1;
	END_IF
	IF angelblue_var = TRUE THEN
		cocktail_var := angelblue;
		angelblue_var := FALSE;
		Anzahl_Cocktails [angelblue] := Anzahl_Cocktails [angelblue] + 1;
	END_IF
	IF brassmonkey_var = TRUE THEN
		cocktail_var := brassmonkey;
		brassmonkey_var := FALSE;
		Anzahl_Cocktails [brassmonkey] := Anzahl_Cocktails [brassmonkey] + 1;
	END_IF
	IF kiba_var = TRUE THEN
		cocktail_var := kiba;
		kiba_var := FALSE;
		Anzahl_Cocktails [kiba] := Anzahl_Cocktails [kiba] + 1;
	END_IF
	IF rumcola_var = TRUE THEN
		cocktail_var := rumcola;
		rumcola_var := FALSE;
		Anzahl_Cocktails [rumcola] := Anzahl_Cocktails [rumcola] + 1;
	END_IF
	IF gintonic_var = TRUE THEN
		cocktail_var := gintonic;
		gintonic_var := FALSE;
		Anzahl_Cocktails [gintonic] := Anzahl_Cocktails [gintonic] + 1;
	END_IF
	IF bluelagoon_var = TRUE THEN
		cocktail_var := bluelagoon;
		bluelagoon_var := FALSE;
		Anzahl_Cocktails [bluelagoon] := Anzahl_Cocktails [bluelagoon] + 1;
	END_IF
	IF osaft_var = TRUE THEN
		cocktail_var := osaft;
		osaft_var := FALSE;
		Anzahl_Cocktails [osaft] := Anzahl_Cocktails [osaft] + 1;
	END_IF
	IF cola_var = TRUE THEN
		cocktail_var := cola;
		cola_var := FALSE;
		Anzahl_Cocktails [cola] := Anzahl_Cocktails [cola] + 1;
	END_IF
	IF banane_var = TRUE THEN
		cocktail_var := banane;
		banane_var := FALSE;
		Anzahl_Cocktails [banane] := Anzahl_Cocktails [banane] + 1;
	END_IF
	IF tonic_var = TRUE THEN
		cocktail_var := tonic;
		tonic_var := FALSE;
		Anzahl_Cocktails [tonic] := Anzahl_Cocktails [tonic] + 1;
	END_IF
	IF sprite_var = TRUE THEN
		cocktail_var := sprite;
		sprite_var := FALSE;
		Anzahl_Cocktails [sprite] := Anzahl_Cocktails [sprite] + 1;
	END_IF
	IF zufallscocktail_var = TRUE THEN
		cocktail_var := zufallscocktail;
		zufallscocktail_var := FALSE;
		Anzahl_Cocktails [zufallscocktail] := Anzahl_Cocktails [zufallscocktail] + 1;
	END_IF
END_PROGRAM
```

#### Init.st
```iecst
PROGRAM _INIT
	cocktail_started := TRUE;

	cocktail_var := 0;
END_PROGRAM
```

- Visualisation Logical/mappView (not shown)

### Program Logical/Zufall (IEC)

#### Variables.var
```iecst
VAR
	Random_Number : ARRAY[1..20] OF USINT; (*Array der Zufallszahlen*)
	m : USINT; (*Hilfsvariable*)
	i : USINT; (*Hilfsvariable*)
	Number_Counter : ARRAY[1..10] OF USINT; (*Zählt, wie oft die Zutaten jeweils vertreten sind*)
	zutat_Menge : ARRAY[1..10] OF UINT;
	zutat_JaNein : ARRAY[1..10] OF BOOL;
	ml : USINT;
	cycle_counter : LREAL; (*Anzahl der durchlaufenen Zyklen zählen*)
	access_counter : USINT; (*Kontrollvariable für Tests, Zählt Anzahl Zugriffe auf Mengenarray bei Mengenbestimmung*)
	k : USINT; (*Hilfsvariable*)
	n : USINT; (*Hilfsvariable*)
	p : USINT; (*Hilfsvariable*)
	q : USINT; (*Hilfsvariable*)
	r : USINT; (*Hilfsvariable*)
	ml_ausgabe : UINT; (*Nur Informationsvariable, um zu testen, wieviele ml am ende tatsächlich rauskommen*)
	menge_alkohol : UINT; (*zum Filtern von Ausreißern*)
	menge_alkoholfrei : UINT; (*zum Filtern von Ausreißern*)
END_VAR
```

#### Cyclic.st
```iecst
PROGRAM _CYCLIC
	IF zufallscocktail_var = FALSE THEN
			//willkürliches Verrechnen zum Erstellen eines Zufalls
			Random_Number[01] := (Random_Number[01] + 73) * ((Random_Number[17] + 1) MOD 14);
			Random_Number[02] := (Random_Number[09] + 73) * ((Random_Number[12] + 1) MOD 16);
			Random_Number[03] := (Random_Number[13] + 73) * ((Random_Number[20] + 1) MOD 11);
			Random_Number[04] := (Random_Number[18] + 73) * ((Random_Number[09] + 1) MOD 17);
			Random_Number[05] := (Random_Number[08] + 73) * ((Random_Number[16] + 1) MOD 19);
			Random_Number[06] := (Random_Number[20] + 72) * ((Random_Number[09] + 1) MOD 13);
			Random_Number[07] := (Random_Number[07] + 73) * ((Random_Number[01] + 1) MOD 17);
			Random_Number[08] := (Random_Number[11] + 73) * ((Random_Number[18] + 1) MOD 18);
			Random_Number[09] := (Random_Number[19] + 73) * ((Random_Number[12] + 1) MOD 11);
			Random_Number[10] := (Random_Number[12] + 73) * ((Random_Number[07] + 1) MOD 16);
			Random_Number[11] := (Random_Number[04] + 73) * ((Random_Number[02] + 1) MOD 10);
			Random_Number[12] := (Random_Number[03] + 73) * ((Random_Number[10] + 1) MOD 19);
			Random_Number[13] := (Random_Number[16] + 73) * ((Random_Number[15] + 1) MOD 18);
			Random_Number[14] := (Random_Number[06] + 73) * ((Random_Number[14] + 1) MOD 17);
			Random_Number[15] := (Random_Number[15] + 73) * ((Random_Number[04] + 1) MOD 15);
			Random_Number[16] := (Random_Number[05] + 73) * ((Random_Number[05] + 1) MOD 10);
			Random_Number[17] := (Random_Number[10] + 73) * ((Random_Number[06] + 1) MOD 18);
			Random_Number[18] := (Random_Number[14] + 73) * ((Random_Number[03] + 1) MOD 14);
			Random_Number[19] := (Random_Number[17] + 73) * ((Random_Number[19] + 1) MOD 19);
			Random_Number[20] := (Random_Number[02] + 73) * ((Random_Number[11] + 1) MOD 16);
			// MOD2: Durchschnittlich 2,6 Zutaten pro Cocktail
			FOR i := 1 TO 4 DO		//Zutatjanein setzen für nicht-alkoholische, Zählen
				IF Random_Number[i] MOD 3 = 0 THEN	//durch MOD 2 häufiger als alkoholische
					zutat_JaNein[i] := TRUE;
					Number_Counter[i] := Number_Counter[i] + 1;
				ELSE
					zutat_JaNein[i] := FALSE;
				END_IF
			END_FOR;
			// MOD4: Durchschnittlich 2,6 Zutaten pro Cocktail
			FOR i := 5 TO 10 DO		//Zutatjanein setzen für alkoholische, Zählen
				IF Random_Number[i] MOD 7 = 0 THEN		//durch MOD 4 weniger häufig als nich-alkoholische
					zutat_JaNein[i] := TRUE;
					Number_Counter[i] := Number_Counter[i] + 1;
				ELSE
					zutat_JaNein[i] := FALSE;
				END_IF
			END_FOR;

			ml := 30;		//Menge zurücksetzen
			ml_ausgabe := 0; //Ausgabemenge zurücksetzen
			FOR i := 1 TO 10 DO		//Mengenarray zurücksetzen
				zutat_Menge[i] := 0;
			END_FOR;

			REPEAT 			//Festlegen der Getränkemengen, zweimal durchgehen
				//über Modulo Werte aufnehmen, Multiplizieren und in zutat_Menge Array schreiben
				IF n MOD 2 = 0 THEN		//es wird immer zwischen den einstelligen und zweistelligen Zufallszahlen gewechselt
					p := 10;
				ELSIF n MOD 3 = 0 THEN
					r := 87;		//alles mit r ist nur, um etwas mehr Zufall zu erzeugen
				ELSE
					p := 0;
					r := 0;
				END_IF
				//Mengen durch unterschiedliche Modulo unterschiedlich festlegen
				FOR i := 1 TO 4 DO
					IF zutat_JaNein[i] = TRUE THEN
						//	m := ml/2;		//m enthält Anteil, der noch aufgefüllt werden muss, hier kann durchschnittliche Menge angepasst werden
						k := (Random_Number[i+p]+r) MOD (ml);		//mit übriger Menge modulo rechnen, sodass maximale Menge nie überschritten
						zutat_Menge[i] := zutat_Menge[i] + k * 10;
						ml := ml - k;
						access_counter := access_counter + 1;		//nur Informationsgewinnung
					END_IF
				END_FOR;
				FOR i := 5 TO 10 DO
					IF zutat_JaNein[i] = TRUE THEN
						m := ml/3;
						k := (Random_Number[i+p]+r) MOD (m);
						zutat_Menge[i] := zutat_Menge[i] + k * 10;
						ml := ml - k;
						access_counter := access_counter + 1;		//nur Informationsgewinnung
					END_IF
				END_FOR;
				n := n + 1;		//Durchläufe der Schleife zählen

				UNTIL
				ml <= 3 OR n > 20 // Die Schleife wird verlassen, wenn ml <= 3 oder wenn zu viele Iterationen stattfinden
			END_REPEAT;
			n := 0;
			REPEAT    //zu allen Zutatenmengen gleichmäßig etwas addieren, sodass Menge erfüllt wird
				FOR i := 10 TO 1 BY -1 DO
					IF i < 5 THEN
						q := 2;
					ELSE
						q := 1;
					END_IF
					IF ml > 1 AND zutat_JaNein[i] = TRUE THEN
						zutat_Menge[i] := zutat_Menge[i] + q*10;
						ml := ml - q;
					END_IF
				END_FOR
				n:= n + 1;
				UNTIL ml <= 1 OR n > 20
			END_REPEAT;

			FOR i:= 1 TO 10 DO		//zur Kontrolle, wieviel letztendlich rauskommt
				ml_ausgabe := ml_ausgabe + zutat_Menge[i];
			END_FOR;
		END_IF
		menge_alkohol := 0;
		menge_alkoholfrei := 0;
		FOR i := 1 TO 4 DO
			menge_alkoholfrei := menge_alkoholfrei + zutat_Menge[i];
		END_FOR
		FOR i := 5 TO 10 DO
			menge_alkohol := menge_alkohol + zutat_Menge[i];
		END_FOR

		IF menge_alkohol <= 280 AND menge_alkoholfrei <= 280 THEN
			FOR i := 1 TO 10 DO
				zutat_Menge_ok[i] := zutat_Menge[i];
				zutat_JaNein_ok[i] := zutat_JaNein[i];
			END_FOR;
		END_IF

		cycle_counter := cycle_counter + 1;		//nur zur Informationsgewinnung
END_PROGRAM
```

### Library Logical/Library (IEC)

#### Library.fun - Exported functions and function blocks
```iecst
{REDUND_ERROR} FUNCTION PumpeOrangensaft : BOOL (*TODO: Hier einen Kommentar eingeben*) (*$GROUP=User,$CAT=User,$GROUPICON=User.png,$CATICON=User.png*)
END_FUNCTION
```

#### PumpeOrangensaft.st - not listed in the package file held
```iecst
(* Frag nicht was für Saft: Einfach Orangensaft *)
FUNCTION PumpeOrangensaft

END_FUNCTION
```

Listed in the project but not available here: Logical/Global.typ, Logical/Libraries, Logical/Library/Types.typ, Logical/Library/Constants.var
